(* Schneider Machine Expert - Basic project Motor_Start/Stop, file version 3.0.0.0 *)
(* ProjectInformations: Name=Motor_Start/Stop *)

HARDWARE
  Cpu 0: TM221CE16T
  EthernetConfiguration: NetworkName=M221, IpAllocationMode=ByDhcp, IpAddress=192.168.1.10, SubnetMask=255.255.255.0
  SerialLineConfiguration: Baud=Baud19200, Parity=ParityEven, DataBits=DataBits8, StopBits=StopBits1, PhysicalMedium=PhysicalMediumRs485, TransmissionMode=TransmissionModeModbusRtu, SlaveId=1, Addressing=SlaveAddressing
  MastTask: UsePeriodScanMode=false, PeriodScan=100
  FastTask: Period=255
  CpuBehavior: StartingMode=StartAsPreviousState, AutoSaveRamOnEeprom=true, WatchdogPeriod=250

SYMBOLS  (address, symbol, comment, settings)
  %M0       TMR_DONE  "Timer done flag"
  %TM0        [Preset=5, Base=OneSecond]
  %I0.0     START_M1
  %I0.1     STOP_M1
  %I0.4     ESTOP
  %Q0.0     MOTOR1

POU Main Program
  (* SectionNumber=1 *)

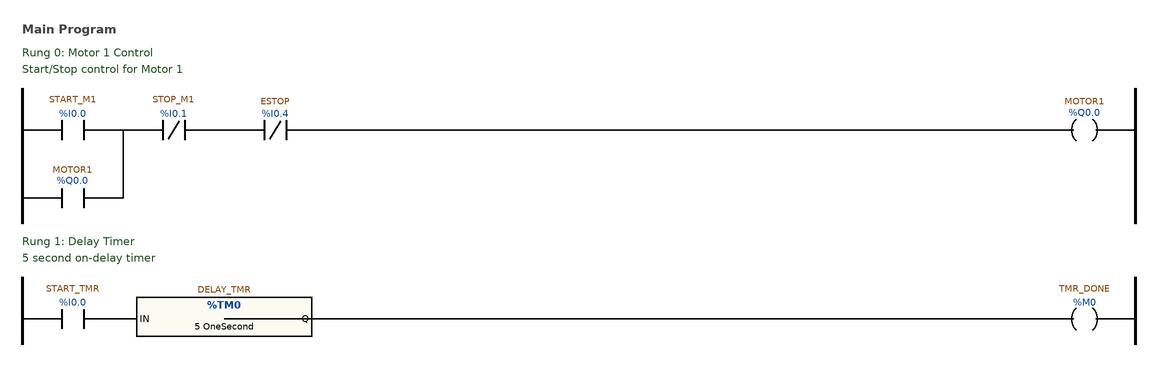

// Rung 0: Motor 1 Control
// Start/Stop control for Motor 1
  LD %I0.0                (* START_M1 *)
  OR %Q0.0                (* MOTOR1 *)
  ANDN %I0.1              (* STOP_M1 *)
  ANDN %I0.4              (* ESTOP *)
  ST %Q0.0                (* MOTOR1 *)
  // as ST:
  //   MOTOR1 := (START_M1 OR MOTOR1) AND NOT STOP_M1 AND NOT ESTOP;

// Rung 1: Delay Timer
// 5 second on-delay timer
  BLK %TM0
  LD %I0.0                (* START_M1 *)
  IN
  OUT_BLK
  LD Q
  ST %M0                  (* TMR_DONE *)
  END_BLK
  // as ST:
  //   %TM0(IN := START_M1);
  //   TMR_DONE := %TM0.Q;
